Staubli VAL3: Socket1.dtx

public bool bCalibrating
public bool bTaskDetOK
num nLatchedValue[10]
public num nMaxNumOfObject = 10
public num nNumOfPart = -1
num nObjectID[10]
  [0] = -1
  [1] = -1
  [2] = -1
  [3] = -1
  [4] = -1
  [5] = -1
  [6] = -1
  [7] = -1
  [8] = -1
  [9] = -1
sio skFromRobot = {link=Socket\fromRobot_sk1}
string sDetNum = "DET0"
string sErrorCode[6]
  [1] = "Could not convert to num ID"
  [2] = "Could not convert to num X"
  [3] = "Could not convert to num Y"
  [4] = "Could not convert to num RZ"
  [5] = "Could not convert to num Encoder Latched Value"
string sTASK = "detect0"
trsf trObjectPos[10]
